TYPE U_SelectorSwitch :
UNION
	IO :ST_SelectorSwitchIO;
	Pos	:E_SelectorSwitchPos;
END_UNION
END_TYPE

(* stored: Version 1.1.0.1
   DUT U_SelectorSwitch: Id {adaacf73-0095-4c3a-a1d8-eb9d456a7bbe} *)
